RoboDK station: ejercicioRobotFiguras.rdk

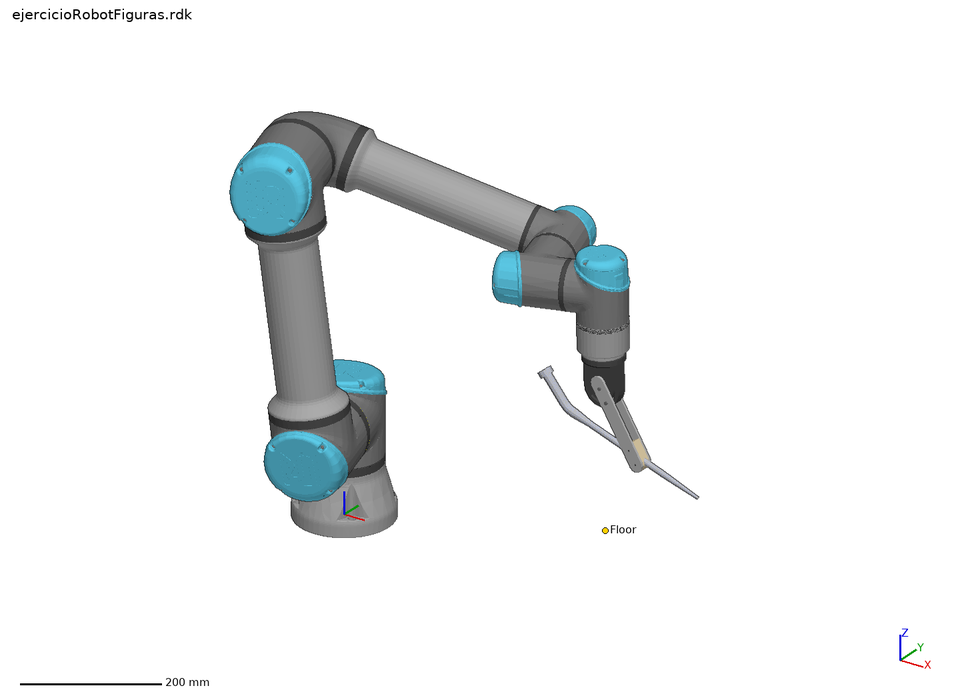
[picture v0: the station drawn from its stored meshes, robots at their saved joint values, targets as dots, program paths as lines]
Station ejercicioRobotFiguras (saved by RoboDK 6.0.4). Poses are relative to the parent item; angles as X-Y-Z fixed-axis rotations.
  - frame UR5e Base at (0, 0, 0) mm
    - robot UR5e: 6 axes, payload 5 kg, reach 850 mm, repeatability 0.03 mm, weight 18.4 kg
        modified DH rows (alpha deg, a mm, theta deg, d mm): 0, 0, 0, 162.5; 90, 0, 180, 0; 0, 425, 0, 0; 0, 392.25, 0, 133.3; -90, 0, 0, 99.7; 90, 0, 180, 99.6
        joint limits [-360, -360, -360, -360, -360, -360] to [360, 360, 360, 360, 360, 360]; home [0, -90, -90, 0, 90, 0]; saved at [17.23, -83, -112.71, -73.5, 90, -72.77]
      - tool Generic Dispenser, TCP at (161.74, 0, 185.22) mm, rotated rx 0 ry 70 rz 0 deg, size 272.6 x 63.8 x 187.1 mm
    - target Floor (Cartesian target) at (450.02, 0, 100) mm, rotated rx 180 ry 0 rz 0 deg; joints [17.23, -83.79, -112.71, -73.5, 90, -72.77] of UR5e
  - Python program Prog1 (listed below)

--- Python program Prog1 ---
Cilindros usando lineas:
# Importamos Librerias
from robodk.robolink import *
from robodk.robomath import *

#Crear Instancia de la Clase RoboLink
rLink = Robolink()

#Obtenemos el Robot selecionado
Robot = rLink.Item('',ITEM_TYPE_ROBOT)

#Vincular variables de Python con targets
varHome = rLink.Item('Home')
varSuelo = rLink.Item('Floor')


# Comprovar el movimiento del robot.
Robot.MoveL(varHome)
Robot.MoveL(varSuelo)

#Obtener la Posicion de Referencia (Pose)
PosRef = varSuelo.Pose()
PosRefAltura = varHome.Pose()

#Pedirle al Usuario Ingrese Vertices.
#Vertices = int(mbox('Ingrese Numero de Vertices: ',entry=True))
Vertices = 360

# Crear Forma Geometria en el Plano.
for i in range(Vertices + 1):
    Angulo = i * 2 * pi / (Vertices)     #Convierte a grados
    Posei = PosRef * rotz(Angulo) * transl(100,0,0) * rotz(-Angulo)
    PoseiAlt= PosRefAltura*rotz(Angulo)*transl(100,0,0)*rotz(-Angulo)
    # Pasar como parametro al movimiento del Robot
    Robot.MoveL(Posei)

    #Proyecta Linea al plano alterno (Altura)
    Robot.MoveL(PoseiAlt)

    # Regresa al Plano Original (Suelo)
    Robot.MoveL(Posei)

Eje_Z = 0
# Crear Forma Geometria en el Plano.
for i in range (50):
    for i in range(Vertices + 1):
        Angulo = i * 2 * pi / (Vertices)     #Convierte a grados
        Posei = PosRef * rotz(Angulo) * transl(100,0,Eje_Z) * rotz(-Angulo)
        Eje_Z = Eje_Z - 0.01

        # Dibuja la trayectoria mediante el movimiento del Robot
        Robot.MoveL(Posei)
Robot.MoveL(varHome)
